{attribute 'qualified_only'}
VAR_GLOBAL
	DateStart : STRING ;
	DateEnd : STRING ;
END_VAR

(* stored: Version 1.1.0.1, ProductVersion 3.1.4024.12
   GVL GVL_HMI: Id {e1899da3-2bcf-4c7c-9527-f9d7395f5218} *)
